# EPICS autosave request: mcaApp/Db/icb_hvps_settings.req
# FILE... icb_hvps_settings.req
# USAGE.. icb_hvps.db fields autosave'd.
$(P)$(HVPS)VOLT_OUT
$(P)$(HVPS)VOLT_LIM
$(P)$(HVPS)INH_LEVEL
$(P)$(HVPS)LATCH_INH
$(P)$(HVPS)LATCH_OVL
$(P)$(HVPS)FRAMP
